(* CODESYS project IoDrvTemplate.library
   Version: 3.5.7.0
   Author: 3S - Smart Software Solutions GmbH
   Description: Template for an IO-driver written in IEC:
      Examples:
      - Bitfield
      - I/O Channels
      - Parameters
      - Diagnostic message and Acknowledge
      - Background diagnosis
      - CAA Device Diagnosis (incl. Reconfigure)
   Title: IoDrvTemplate
   DocFormat: reStructuredText
   DefaultNamespace: TPL
   LanguageModelAttribute: qualified-access-only
   Company: MyCompany
   Placeholder: IoDrvTemplate

Project tree, tasks and I/O mapping:
  libraries: SysMem, * (System); SysCpuHandling, * (System); IoDrvBase, * (System); IoStandard, * (System); IoDriver Parameter Interfaces, * (System); Base Interfaces, * (System); IoDriver Interfaces, * (System); CmpErrors2 Interfaces, * (System); SysTypes2 Interfaces, * (System); CAA Device Diagnosis, 3.5.8.0 (CAA Technical Workgroup); CAA Types Extern, * (CAA Technical Workgroup); CmpAsyncMgr, * (System)
  function block IoDrvTemplate [ST]: IoDrvWriteParameter, IoDrvReadParameter, IoDrvReadInputs, IoDrvIdentify, IoDrvUpdateConfiguration, IoDrvWatchdogTrigger, IoDrvScanModules, IoDrvUpdateMapping, IoDrvWriteOutputs, IoDrvStartBusCycle, IoDrvGetModuleDiagnosis, QueryInterface, FB_Reinit, Initialize, FB_Exit, FB_Init, IoDrvGetConnector, Cleanup, FreeScanData
  function block IoDrvTemplateDiag [ST]: ChildNodeCount, Connector, Enable, FirstChildNode, Index, IsRootNode, NextSiblingNode, ParentNode, SiblingNodeCount, GetChild, Initialize_Diag, GetSpecificDeviceState, SetCommunicationState, GetDeviceInfo, GetDeviceErrorAsync, GetSpecificDeviceErrorAsync, GetDeviceDiagnosisInfo, GetDeviceState, CheckCurrentSupportedCommunicationState, CheckSupportedCommunicationState, GetLogger, GetBusScanAsync, GetQoS, GetBusErrorAsync, GetBusDiagnosisInfo, GetBusState, GetBusInfo, GetSpecificBusState, ReconfigureActive, SiblingIRP, ReconfigureAsync, RegisterIRPChild
  Functions/
    function IsConnectorEnabled [ST]
  global variables GVL
*)

// GVL
VAR_GLOBAL
	g_stComponentName : STRING := 'IoDrvTemplate';
END_VAR

// IoDrvTemplate
{attribute 'no_assign'}
{attribute 'conditionalshow_all_locals' := 'IoDrvDebug'}
FUNCTION_BLOCK IoDrvTemplate EXTENDS IoDrvBase IMPLEMENTS ICmpIoDrvParameter
VAR_INPUT
END_VAR
VAR_OUTPUT
END_VAR
VAR CONSTANT
	CLASSID_CCmpIoDrvTemplate : DWORD := 16#0000FF02;
	IOSize : DWORD := 5;
END_VAR
VAR
	_byInputs : ARRAY [0..IOSize-1] OF BYTE;
	_byOutputs : ARRAY [0..IOSize-1] OF BYTE;
	_IIoDrv : ICmpIoDrv;
	_IIoDrvParameter : ICmpIoDrvParameter;
	_xBackGroundDiagStarted : BOOL;
	_bDeactivated : BOOL;
	
	//Variables for scan
	_iScannedSlaves : INT;
	_pScanList : POINTER TO IoStandard.IoConfigConnector;
END_VAR

{attribute 'conditionalshow' := 'IoDrvDebug'}
METHOD IoDrvWriteParameter : UDINT
VAR_INPUT
	pConnector : POINTER TO IoConfigConnector;
	pParameter : POINTER TO IoConfigParameter;
	pData : POINTER TO BYTE;
	dwBitSize : DWORD;
	dwBitOffset : DWORD;
END_VAR
VAR
	pParam : POINTER TO IoConfigParameter;
	pstDiagString : POINTER TO STRING;
	pValue : POINTER TO BYTE;
END_VAR
IF pConnector = 0 OR pParameter = 0 OR pData = 0 THEN
	IoDrvWriteParameter := Errors.ERR_PARAMETER;
	RETURN;	
END_IF

//If IoDrvWriteParameter returns a value unequal ERR_OK, write parameter will be handled by the IO-manager!
//Note: Code must be only implemented here if there are special things to do.

IoDrvWriteParameter := Errors.ERR_OK;

CASE pParameter^.dwParameterId OF
	393221: //simulate diag
		IF pData^ <> 0 THEN
			(*
				Example for extended Diagnostic:
				- here a string value is written to parameter of channeltype "diag": when "CF_CONNECTOR_DIAGNOSTIC_AVAILABLE" is set in the connector, the diagnostic message is read with ReadParameter.
			*)
			pParam := IoMgrConfigGetParameter(pConnector, 4711);
			IF pParam <> 0 THEN
				pstDiagString := IoMgrConfigGetParameterValuePointer(pParam, 0);
				IF pstDiagString <> 0 THEN
					pstDiagString^ := 'Error pending';
				END_IF
			END_IF
			
			(*
				set diagnostic available flag to trigger reading of diagnosis parameter
			*) 
			IoMgrConfigSetDiagnosis(pConnector, Connectorflags.CF_CONNECTOR_DIAGNOSTIC_AVAILABLE);
		END_IF
		RETURN;
	393222, 393223:
		//here you can add some special code for the three parameters
		pValue := pParameter^.dwValue;
		SysMemCpy((pValue + dwBitOffset/8), pData, MIN(DWORD_TO_BYTE(dwBitSize/8), UINT_TO_BYTE(pParameter^.wLen / 8)));			
		RETURN;
	4712: 
		(*
				Example for extended Diagnostic Acknowledge:
				- Parameter needs channel type "diagack": when user presses ACKNOWLEDGE WriteParameter is called
				- here only the flag is reset, so the diag message is not shown in the Editor any more  
		*)
		IoMgrConfigResetDiagnosis(pConnector, Connectorflags.CF_CONNECTOR_DIAGNOSTIC_AVAILABLE);
		RETURN;
	ELSE
		pValue := pParameter^.dwValue; 
		SysMemCpy(pDest := pValue + dwBitOffset/8, pSrc := pData, pParameter^.wLen / 8);
END_CASE

IoDrvWriteParameter := Errors.ERR_FAILED;
END_METHOD

{attribute 'conditionalshow' := 'IoDrvDebug'}
METHOD IoDrvReadParameter : UDINT
VAR_INPUT
	pConnector : POINTER TO IoConfigConnector;
	pParameter : POINTER TO IoConfigParameter;
	pData : POINTER TO BYTE;
	dwBitSize : DWORD;
	dwBitOffset : DWORD;
END_VAR
VAR
	pValue : POINTER TO BYTE;
END_VAR
IF 	pConnector = 0 OR pParameter = 0 OR pData = 0 THEN
	IoDrvReadParameter := Errors.ERR_PARAMETER;
	RETURN;	
END_IF

IoDrvReadParameter := Errors.ERR_OK;

pValue := pParameter^.dwValue;
IF pValue <> 0 THEN
	CASE pParameter^.dwParameterId OF
		4711: 
			(*
				Example for extended Diagnostic:
				- Parameter needs channel type "diag": as long as connectorflag "CF_CONNECTOR_DIAGNOSTIC_AVAILABLE" is set, the IoDrvReadParameter will be called with the Parameter of channeltype "diag"
				- One may return a string that is shown in "status" editor in CODESYS			
			*)

			IF pParameter^.wLen >= (dwBitOffset + dwBitSize) THEN	 
				SysMemCpy(pData, (pValue + dwBitOffset/8), MIN(DWORD_TO_BYTE(dwBitSize/8), UINT_TO_BYTE(pParameter^.wLen / 8)));		
				RETURN;
			END_IF
		ELSE
			// handle other parameters here: be aware of length of destination buffer
			SysMemCpy(pData, pValue + dwBitOffset/8, MIN(DWORD_TO_BYTE(dwBitSize/8), UINT_TO_BYTE(pParameter^.wLen / 8)));
			RETURN;
	END_CASE
END_IF
// All standard parameters of our device are handled by the IO-manager!
IoDrvReadParameter := Errors.ERR_FAILED;
END_METHOD

{attribute 'conditionalshow' := 'IoDrvDebug'}
METHOD IoDrvReadInputs : UDINT
VAR_INPUT
	pConnectorMapList : POINTER TO IoConfigConnectorMap;
	nCount : DINT;
END_VAR
VAR
	i,j : DINT;
	wSize : WORD;
	pConnectorMap : POINTER TO IoStandard.IoConfigConnectorMap;
	pChannelMap : POINTER TO IoStandard.IoConfigChannelMap;
	pbyIecAddress : POINTER TO BYTE;
	bySrcValue : BYTE;
	bySrcMask : BYTE;
	wSrcIndex : WORD;	
	wDestIndex : WORD;	
END_VAR
IoDrvReadInputs_Count := IoDrvReadInputs_Count + 1;

IF _bDeactivated THEN
	RETURN;
END_IF

IF pConnectorMapList = 0 OR nCount = 0 THEN
	IoDrvReadInputs := Errors.ERR_PARAMETER;
	RETURN;
END_IF

FOR i:=0 TO nCount - 1 DO
	pConnectorMap := ADR(pConnectorMapList[i]);
	
	FOR j:= 0 TO UDINT_TO_UINT(pConnectorMap^.dwNumOfChannels) - 1 DO
		pChannelMap := ADR(pConnectorMap^.pChannelMapList[j]);
		
		// input medium byteorder: Little Endian:		
		IoMgrCopyInputLE(pChannelMap, pChannelMap^.pParameter^.dwDriverSpecific);
		
		// input medium byteorder: Big Endian:		
		//IoMgrCopyInputBE(ADR(pChannelMap, pChannelMap^.pParameter^.dwDriverSpecific);
	END_FOR
END_FOR

IoDrvReadInputs := Errors.ERR_OK;
END_METHOD

{attribute 'conditionalshow' := 'IoDrvDebug'}
METHOD IoDrvIdentify : UDINT
VAR_INPUT
	pConnector : POINTER TO IoConfigConnector;	
END_VAR
VAR
END_VAR
IoDrvIdentify_Count := IoDrvIdentify_Count + 1;
IoDrvIdentify := Errors.ERR_NOTIMPLEMENTED;
END_METHOD

{attribute 'conditionalshow' := 'IoDrvDebug'}
METHOD IoDrvUpdateConfiguration : UDINT
VAR_INPUT
	pConnectorList : POINTER TO IoConfigConnector;
	nCount : DINT;
END_VAR
VAR
	pParameter : POINTER TO IoConfigParameter;	
	pChild : POINTER TO IoConfigConnector;	
	pstConnectorVendorName : POINTER TO STRING;
	pstConnectorDeviceName : POINTER TO STRING;
	dwTest : DWORD;
	Result : RTS_IEC_RESULT;
END_VAR
IoDrvUpdateConfiguration_Count := IoDrvUpdateConfiguration_Count + 1;
IoDrvUpdateConfiguration := Errors.ERR_OK;

IF pConnectorList = 0 THEN
	// Reset application
	m_pConnector^.hIoDrv := 0; // no callbacks from runtime!
	m_pConnector^.pFather^.hIoDrv := 0;
	Cleanup();
	RETURN;
END_IF

m_pConnector := IoMgrConfigGetConnector(pConnectorList, ADR(nCount), m_wModuleType, m_dwInstance);

IF m_pConnector = 0 THEN
	IoDrvUpdateConfiguration := ERRORS.ERR_PARAMETER;
	RETURN;
END_IF

//check if device is enabled in the device tree
_bDeactivated := NOT IsConnectorEnabled(m_pConnector);

IF m_pConnector^.hIoDrv = 0 THEN
	//always needed for reconfigure!
	m_pConnector^.hIoDrv := m_hInterface;
	m_pConnector^.pFather^.hIoDrv := m_hInterface;
END_IF

IF _bDeactivated THEN
	IoDrvUpdateConfiguration := CmpErrors.Errors.ERR_OK;
	RETURN;
END_IF

IF m_pConnector^.hIoDrv = m_hInterface THEN
	{IF defined (pou:IoMgrConfigSetDiagnosis)}
	IoMgrConfigSetDiagnosis(m_pConnector,
							ConnectorFlags.CF_DRIVER_AVAILABLE OR
							ConnectorFlags.CF_CONNECTOR_FOUND OR
							ConnectorFlags.CF_CONNECTOR_CONFIGURED OR
							ConnectorFlags.CF_CONNECTOR_ACTIVE);
	{END_IF}
	
	{IF defined (pou:IoMgrConfigSetDiagnosis)}
	IoMgrConfigSetDiagnosis(m_pConnector^.pFather,
							ConnectorFlags.CF_DRIVER_AVAILABLE OR
							ConnectorFlags.CF_CONNECTOR_FOUND OR
							ConnectorFlags.CF_CONNECTOR_CONFIGURED OR
							ConnectorFlags.CF_CONNECTOR_ACTIVE);
	{END_IF}

	{IF defined (pou:IoMgrSetDriverProperties)}			
		IoMgrSetDriverProperties(m_hInterface, DRVPROP_CONSISTENCY OR DRVPROP_BACKGROUND_GETDIAG);
		//Note: background diagnosis property flag is optional (supported with 3.5.1.0 runtime)
	{END_IF}										

	//Read some parameters
	pParameter := IoMgrConfigGetParameter(m_pConnector, 393218);
	IF pParameter <> 0 THEN
		pstConnectorVendorName := IoMgrConfigGetParameterValuePointer(pParameter, ADR(Result));
	END_IF
	pParameter := IoMgrConfigGetParameter(m_pConnector, 393219);
	IF pParameter <> 0 THEN
		pstConnectorDeviceName := IoMgrConfigGetParameterValuePointer(pParameter, ADR(Result));
	END_IF
	pParameter := IoMgrConfigGetParameter(m_pConnector, 393220);	(* test parameter *)
	IF (pParameter <> 0) THEN
		dwTest := IoMgrConfigGetParameterValueDword(pParameter, ADR(Result));	(* Test parameter value *)			
	END_IF
	
	//Setup I/O area
	pParameter := IoMgrConfigGetParameter(m_pConnector, 1000);		(* inputs *)
	IF (pParameter <> 0) THEN
		pParameter^.dwDriverSpecific := ADR(_byInputs[0]);					(* Device offset 0 *)
	END_IF
	pParameter := IoMgrConfigGetParameter(m_pConnector, 1001);		(* inputs *)
	IF (pParameter <> 0) THEN
		pParameter^.dwDriverSpecific := ADR(_byInputs[4]);					(* Device offset 0 *)
	END_IF
	pParameter := IoMgrConfigGetParameter(m_pConnector, 2000);		(* outputs *)
	IF (pParameter <> 0) THEN
		pParameter^.dwDriverSpecific := ADR(_byOutputs[0]);					(* Device offset 0 *)
	END_IF
	pParameter := IoMgrConfigGetParameter(m_pConnector, 2001);		(* outputs *)
	IF (pParameter <> 0) THEN
		pParameter^.dwDriverSpecific := ADR(_byOutputs[4]);					(* Device offset 0 *)
	END_IF
	
	//Go through all childs of the device
	pChild := IoMgrConfigGetFirstChild(m_pConnector, ADR(nCount), m_pConnector);
	WHILE (pChild <> 0) DO
		IF IsConnectorEnabled(pChild) THEN
			pChild^.hIoDrv := m_hInterface;	
			{IF defined (pou:IoMgrConfigSetDiagnosis)}
			IoMgrConfigSetDiagnosis(pChild,
									ConnectorFlags.CF_DRIVER_AVAILABLE OR
									ConnectorFlags.CF_CONNECTOR_FOUND OR
									ConnectorFlags.CF_CONNECTOR_CONFIGURED OR
									ConnectorFlags.CF_CONNECTOR_ACTIVE);
			{END_IF}
		END_IF
		pChild := IoMgrConfigGetNextChild(pChild, ADR(nCount), m_pConnector);
	END_WHILE
END_IF
END_METHOD

{attribute 'conditionalshow' := 'IoDrvDebug'}
METHOD IoDrvWatchdogTrigger : UDINT
VAR_INPUT
	pConnector : POINTER TO IoConfigConnector;	
END_VAR
VAR
END_VAR
IoDrvWatchdogTrigger_Count := IoDrvWatchdogTrigger_Count + 1;
IoDrvWatchdogTrigger := Errors.ERR_OK;
END_METHOD

{attribute 'conditionalshow' := 'IoDrvDebug'}
METHOD IoDrvScanModules : UDINT
VAR_INPUT
	pConnector : POINTER TO IoConfigConnector;
	ppConnectorList : POINTER TO POINTER TO IoConfigConnector;
	pnCount : POINTER TO DINT;	
END_VAR
VAR
	pCurConnector : POINTER TO IoConfigConnector;
	pParameter: POINTER TO IoConfigParameter;
	pString : POINTER TO STRING;
	i : INT;
	j : INT;
END_VAR
IoDrvScanModules_Count := IoDrvScanModules_Count + 1;

IF pConnector = 0 OR ppConnectorList = 0 OR pnCount = 0 THEN
	IoDrvScanModules := Errors.ERR_PARAMETER;
	RETURN;
END_IF

FreeScanData();

pnCount^ := 0;
ppConnectorList^ := 0;

(*
	TODO: implement specific bus scan!
	Note: IoDrvScanModules is called in communication task. If this method takes too long (> 20s) a communication timeout may happen.
	In this cases you can do a segmented scan by setting IoStandard.ConnectorOptions.CO_SCAN_PENDING_SUPPORTED.
	If IoDrvScanModules returns ERR_PENDING method is called again. The results of all calls are combined by the GUI.
*)

(*The following code just generates some example data. The real scan algorithm has to set the values regarding to the scan result. *)
_iScannedSlaves := 2; //we return 2 slaves

IF _iScannedSlaves > 0 THEN
	//Allocate memory for the connector list
	ppConnectorList^ := SysMemAllocData(g_stComponentName, INT_TO_DWORD(_iScannedSlaves * SIZEOF(IoStandard.IoConfigConnector)), 0);
	IF ppConnectorList = 0 THEN
		IoDrvScanModules := Errors.ERR_FAILED;
		_iScannedSlaves := 0;
		RETURN;
	END_IF
	SysMem.SysMemSet(ppConnectorList^, 0, INT_TO_DWORD(_iScannedSlaves * SIZEOF(IoStandard.IoConfigConnector)));
END_IF

pCurConnector := ppConnectorList^;
FOR i := 0 TO _iScannedSlaves - 1 DO
	pCurConnector^.dwNumOfParameters := 4; //we return the 4 mandatory parameters
	//Alocate memory for the parameter list of the current connector
	pCurConnector^.pParameterList := SysMemAllocData(g_stComponentName, pCurConnector^.dwNumOfParameters * SIZEOF(IoStandard.IoConfigParameter), 0);
	SysMem.SysMemSet(pCurConnector^.pParameterList, 0, pCurConnector^.dwNumOfParameters * SIZEOF(IoStandard.IoConfigParameter));
	
    pParameter := pCurConnector^.pParameterList;
	
	//Set parameter: Vendor code
	pParameter^.dwParameterId := 1;
	pParameter^.dwValue := 1; //Vendor Code
	pParameter^.wLen := 32;
	pParameter^.wType := INT_TO_WORD(TypeClass.TYPE_DWORD); //16#4
	pParameter^.dwFlags := IoStandard.PVF_READ OR IoStandard.PVF_WRITE OR IoStandard.PVF_VALUE; //16#34
	
	pParameter := pParameter + SIZEOF(IoStandard.IoConfigParameter);
	
	//Set parameter: Product code
	pParameter^.dwParameterId := 2;
	pParameter^.dwValue := 2; //Product Code
	pParameter^.wLen := 32;
	pParameter^.wType := INT_TO_WORD(TypeClass.TYPE_DWORD); //16#4
	pParameter^.dwFlags := IoStandard.PVF_READ OR IoStandard.PVF_WRITE OR IoStandard.PVF_VALUE; //16#34
	
	pParameter := pParameter + SIZEOF(IoStandard.IoConfigParameter);
	
	//Set parameter: Revision Number
	pParameter^.dwParameterId := 3;
	pParameter^.dwValue := 10; //Revision Number
	pParameter^.wLen := 32;
	pParameter^.wType := INT_TO_WORD(TypeClass.TYPE_DWORD); //16#4
	pParameter^.dwFlags := IoStandard.PVF_READ OR IoStandard.PVF_WRITE OR IoStandard.PVF_VALUE; //16#34
	
	pParameter := pParameter + SIZEOF(IoStandard.IoConfigParameter);
	
	//Set parameter: Device Identification
	pParameter^.dwParameterId := 4;
	pParameter^.dwValue := SysMemAllocData(g_stComponentName, SIZEOF(STRING), 0);
	pString := pParameter^.dwValue;
	pString^ := '1_2_10'; // Device Identification
	pParameter^.wLen := SIZEOF(STRING);
	pParameter^.wType := INT_TO_WORD(TypeClass.TYPE_STRING); //16#10
	pParameter^.dwFlags := IoStandard.PVF_READ OR IoStandard.PVF_WRITE OR IoStandard.PVF_POINTER; //16#32
		
	pCurConnector^.hIoDrv := THIS;
	pCurConnector^.pFather := pConnector;
	pCurConnector^.wType := ConnectorTypes.CT_CAN_SLAVE; //we return a CANopen Slave connector
	
	pCurConnector := pCurConnector + SIZEOF(IoStandard.IoConfigConnector);
END_FOR

pnCount^ := _iScannedSlaves; //Set number of scanned devices
IoDrvScanModules := CmpErrors.Errors.ERR_OK;
END_METHOD

{attribute 'conditionalshow' := 'IoDrvDebug'}
METHOD IoDrvUpdateMapping : UDINT
VAR_INPUT
	pTaskMapList : POINTER TO IoConfigTaskMap;
	nCount : DINT;	
END_VAR
VAR
END_VAR
IoDrvUpdateMapping_Count := IoDrvUpdateMapping_Count + 1;

IF (pTaskMapList = 0) THEN
	IoDrvUpdateMapping := Errors.ERR_PARAMETER;
	RETURN;
END_IF

IoDrvUpdateMapping := Errors.ERR_OK;
END_METHOD

{attribute 'conditionalshow' := 'IoDrvDebug'}
METHOD IoDrvWriteOutputs : UDINT
VAR_INPUT
	pConnectorMapList : POINTER TO IoConfigConnectorMap;
	nCount : DINT;
END_VAR
VAR
	i,j : DINT;
	wSize : WORD;
	pConnectorMap : POINTER TO IoStandard.IoConfigConnectorMap;
	pChannelMap : POINTER TO IoStandard.IoConfigChannelMap;
	pbyIecAddress : POINTER TO BYTE;
	bySrcValue : BYTE;
	wSrcIndex : WORD;	
	bySrcMask : BYTE;
	wDestIndex : WORD;	
END_VAR
IoDrvWriteOutputs_Count := IoDrvWriteOutputs_Count + 1;

IF _bDeactivated THEN
	RETURN;
END_IF

IF pConnectorMapList = 0 OR nCount = 0 THEN
	IoDrvWriteOutputs := Errors.ERR_PARAMETER;
	RETURN;
END_IF

FOR i:=0 TO nCount - 1 DO
	pConnectorMap := ADR(pConnectorMapList[i]);
	
	FOR j:= 0 TO UDINT_TO_UINT(pConnectorMap^.dwNumOfChannels) - 1 DO
		pChannelMap := ADR(pConnectorMap^.pChannelMapList[j]);
		
		// output medium byteorder: Little Endian:		
		IoMgrCopyOutputLE(pChannelMap, pChannelMap^.pParameter^.dwDriverSpecific);
		
		// output medium byteorder: Big Endian:		
		//IoMgrCopyOutputBE(pChannelMap, pChannelMap^.pParameter^.dwDriverSpecific);
	END_FOR
END_FOR

IoDrvWriteOutputs := Errors.ERR_OK;
END_METHOD

{attribute 'conditionalshow' := 'IoDrvDebug'}
METHOD IoDrvStartBusCycle : UDINT
VAR_INPUT
	pConnector : POINTER TO IoConfigConnector;
END_VAR
VAR
END_VAR
IoDrvStartBusCycle_Count := IoDrvStartBusCycle_Count + 1;

IF _bDeactivated OR_ELSE pConnector <> m_pConnector THEN
	RETURN;
END_IF

//if background diagnosis is not active call IoDrvGetModuleDiagnosis; normally it will be called by the runtime if DRVPROP_BACKGROUND_GETDIAG is set
IF NOT _xBackGroundDiagStarted THEN
	IoDrvGetModuleDiagnosis(m_pConnector); //DRVPROP_BACKGROUND_GETDIAG not set or runtime version < V3.5.1.0
END_IF

//optional: call IoDrvWatchdogTrigger or set driver property DRVPROP_WATCHDOG in UpdateConfiguration
IoDrvWatchdogTrigger(pConnector);

//simulate input data (only for test)
MemCpy(ADR(_byInputs), ADR(_byOutputs), IOSize);

IoDrvStartBusCycle := Errors.ERR_OK;
END_METHOD

METHOD IoDrvGetModuleDiagnosis : UDINT
VAR_INPUT
	pConnector : POINTER TO IoConfigConnector;
END_VAR
VAR
END_VAR
IF pConnector = 0 THEN
	//we are called from the background task
	_xBackGroundDiagStarted := TRUE;
END_IF

//Todo: update connectorflags if something changed

IoDrvGetModuleDiagnosis_Count := IoDrvGetModuleDiagnosis_Count + 1;
IoDrvGetModuleDiagnosis := Errors.ERR_NOTIMPLEMENTED;
END_METHOD

{attribute 'conditionalshow' := 'IoDrvDebug'}
METHOD QueryInterface : POINTER TO POINTER TO BYTE
VAR_INPUT
	iid : DWORD; (* InterfaceID *)
	pResult : POINTER TO UDINT;	
END_VAR
VAR
END_VAR
QueryInterface_Count := QueryInterface_Count + 1;
IF iid = ITFID_ICmpIoDrv THEN
	QueryInterface := ADR(_IIoDrv);
	AddRef();
	IF (pResult <> 0) THEN
		pResult^ := Errors.ERR_OK;
	END_IF
	RETURN;	
ELSIF iid = ITFID_ICmpIoDrvParameter THEN
	QueryInterface := ADR(_IIoDrvParameter);
	AddRef();
	IF (pResult <> 0) THEN
		pResult^ := Errors.ERR_OK;
	END_IF	
	RETURN;	
ELSE
	QueryInterface := SUPER^.QueryInterface(iid, pResult);
END_IF
END_METHOD

{attribute 'conditionalshow' := 'IoDrvDebug'}
METHOD FB_Reinit : BOOL
VAR_INPUT
END_VAR
VAR
END_VAR
FB_Reinit_Count := FB_Reinit_Count + 1;
FB_Reinit := TRUE;
END_METHOD

{attribute 'conditionalshow' := 'IoDrvDebug'}
METHOD Initialize : UDINT
VAR_INPUT
	wModuleType : UINT;
	dwInstance : UDINT;
	pConnector : POINTER TO IoConfigConnector; 
END_VAR
VAR
END_VAR
Initialize_Count := Initialize_Count + 1;

m_wModuleType := wModuleType;
m_dwInstance := dwInstance;
m_Info.wModuleType := wModuleType;

Initialize := Errors.ERR_OK;
END_METHOD

{attribute 'conditionalshow' := 'IoDrvDebug'}
METHOD FB_Exit : BOOL
VAR_INPUT
	bInCopyCode: BOOL;	
END_VAR
VAR
END_VAR
FB_Exit_Count := FB_Exit_Count + 1;
FB_Exit := TRUE;
END_METHOD

{attribute 'conditionalshow' := 'IoDrvDebug'}
METHOD FB_Init : BOOL
VAR_INPUT
	bInitRetains: BOOL;
	bInCopyCode: BOOL;
END_VAR
VAR
	Result : UDINT;
END_VAR
FB_Init_Count := FB_Init_Count + 1;

m_Info.szDriverName := 'IoDrvTemplateIEC';
m_Info.szVendorName := 'MyCompany';
m_Info.szDeviceName := 'MyCard';
m_Info.wModuleType := 40100;

_IIoDrv := THIS^;
_IIoDrvParameter := THIS^;

m_IBaseItf := THIS^;
m_hInterface := IoMgrRegisterInstance2(CLASSID_CCmpIoDrvTemplate, m_IBaseItf, ADR(Result));
FB_Init := TRUE;
END_METHOD

{attribute 'conditionalshow' := 'IoDrvDebug'}
METHOD IoDrvGetConnector : POINTER TO IoConfigConnector
VAR_INPUT
	pResult : POINTER TO RTS_IEC_RESULT;
END_VAR
VAR
END_VAR
IF m_pConnector = 0 THEN
	IF pResult <> 0 THEN
		pResult^ := Errors.ERR_FAILED;
	END_IF
	IoDrvGetConnector := 0;	
	RETURN;
END_IF
IF pResult <> 0 THEN
	pResult^ := Errors.ERR_OK;
END_IF
IoDrvGetConnector := m_pConnector;
END_METHOD

{attribute 'conditionalshow' := 'IoDrvDebug'}
METHOD Cleanup
VAR_INPUT
END_VAR
VAR

END_VAR
FreeScanData();
END_METHOD

{attribute 'conditionalshow' := 'IoDrvDebug'}
METHOD FreeScanData
VAR_INPUT
END_VAR
VAR
	pCurConnector : POINTER TO IoConfigConnector;
	pParameter : POINTER TO IoConfigParameter;	
	i : INT;
	j : INT;
END_VAR
//Free device scan data
IF _iScannedSlaves > 0 AND _pScanList <> 0 THEN
	pCurConnector := _pScanList;
	FOR i := 0 TO _iScannedSlaves - 1 DO
		pParameter := pCurConnector^.pParameterList;
		IF pParameter <> 0 THEN
			FOR j := 0 TO DWORD_TO_INT(pCurConnector^.dwNumOfParameters) - 1 DO
				IF (pParameter^.dwFlags AND IoStandard.ParameterValueFlags.PVF_POINTER) = IoStandard.ParameterValueFlags.PVF_POINTER THEN
					// dwValue is pointer
					IF pParameter^.dwValue <> 0 THEN
						SysMemFreeData(g_stComponentName, pParameter^.dwValue);
					END_IF
				END_IF
				pParameter := pParameter + SIZEOF(IoConfigParameter);	
			END_FOR
			SysMemFreeData(g_stComponentName, pCurConnector^.pParameterList);
		END_IF
		pCurConnector := pCurConnector + SIZEOF(IoStandard.IoConfigConnector);
	END_FOR
	SysMemFreeData(g_stComponentName, _pScanList);
	_pScanList := 0;
 	_iScannedSlaves := 0;
END_IF
END_METHOD

END_FUNCTION_BLOCK

// Functions/IsConnectorEnabled
{attribute 'conditionalshow' := '3SLib_Developer'}
FUNCTION IsConnectorEnabled : BOOL
VAR_INPUT
	pConnector : POINTER TO IoStandard.IoConfigConnector;
END_VAR
VAR
END_VAR

{IF defined (variable:CF_DEVICE_ENABLED) AND defined (variable:CF_DIAG_PROVIDER)}
	IF (pConnector^.dwFlags AND IoStandard.ConnectorFlags.CF_DIAG_PROVIDER) <> 0 THEN
		IsConnectorEnabled := (pConnector^.dwFlags AND IoStandard.ConnectorFlags.CF_DEVICE_ENABLED) <> 0;
	ELSE
		IsConnectorEnabled := (pConnector^.dwFlags AND ConnectorFlags.CF_ENABLE) <> 0;
	END_IF
{ELSE}
	IsConnectorEnabled := (pConnector^.dwFlags AND ConnectorFlags.CF_ENABLE) <> 0;
{END_IF}

END_FUNCTION

// IoDrvTemplateDiag
//This function block implements the diagnosis code for CAA Device Diagnosis.
{attribute 'no_assign'}
{attribute 'conditionalshow_all_locals' := 'IoDrvDebug'}
FUNCTION_BLOCK IoDrvTemplateDiag EXTENDS IoDrvTemplate IMPLEMENTS DED.IDevice2, DED.IBus, DED.IStack, DED.IReconfigureProvider
VAR_INPUT
END_VAR
VAR_OUTPUT
END_VAR
VAR
	_diag : DED.CAADiagnosisBase;
	_tree : DED.CAADiagTreeBase;
	_reconfig : DED.CAAReconfigureBase; //optional
END_VAR

(*Returns the number of childs below the current node*)
PROPERTY ChildNodeCount : CAA.COUNT
GET
ChildNodeCount := _tree.ChildNodeCount;
END_GET
END_PROPERTY

PROPERTY Connector : POINTER TO IoStandard.IoConfigConnector
GET
Connector := _tree.Connector;
END_GET
END_PROPERTY

(*This property returns if the node is enabled in the device tree. The setter can be used to change the Enabled flag. If enabling/disabling is not supported on the node the flag’s value will not change.*)
PROPERTY Enable : BOOL
GET
Enable := _tree.Enable;
END_GET
SET
_tree.Enable := Enable;
END_SET
END_PROPERTY

(*Returns the first child node below the current one*)
PROPERTY FirstChildNode : DED.INode
GET
FirstChildNode := _tree.FirstChildNode;
END_GET
END_PROPERTY

PROPERTY Index : UDINT
GET
Index := _tree.Index;
END_GET
SET
_tree.Index := Index;
END_SET
END_PROPERTY

(* returns true, if the current node is the root (plc) node, otherwise false*)
PROPERTY IsRootNode : BOOL
GET
IsRootNode := _tree.IsRootNode;
END_GET
END_PROPERTY

(* returns the next sibling node at the same level
 used for step through all nodes*)
PROPERTY NextSiblingNode : DED.INode
GET
NextSiblingNode := _tree.NextSiblingNode;
END_GET
END_PROPERTY

(* Returns the parent node or zero if already the root node is reached*)
PROPERTY ParentNode : DED.INode
GET
ParentNode := _tree.ParentNode;
END_GET
END_PROPERTY

(* Returns the number of sibling (same level) nodes*)
PROPERTY SiblingNodeCount : CAA.COUNT
GET
SiblingNodeCount := _tree.SiblingNodeCount;
END_GET
END_PROPERTY

{attribute 'hide'}
METHOD GetChild : DED.INode
VAR_INPUT
	udiIndex	: UDINT;
END_VAR
GetChild:= _tree.GetChild(udiIndex);
END_METHOD

{attribute 'hide'}
METHOD Initialize_Diag : UDINT
VAR_INPUT
	pConnector	: POINTER TO IoStandard.IoConfigConnector;
	nConnectorCount	: DINT;
	parent	: POINTER TO DED.INode;
	children	: POINTER TO DED.INode;
	udiChildCount	: UDINT;
END_VAR
//general initialization code: do not remove!
_tree.Initialize_Diag(pConnector, nConnectorCount, parent, children, udiChildCount);
_diag.Initialize_Diag(pConnector, nConnectorCount);

//if IReconfigureProvider is implemented
_reconfig.Initialize_Diag(THIS^);
END_METHOD

{attribute '''NORMAL__COMMENT' := 'Returns the fieldbus specific device state; interpretation is fieldbus dependent'}
(*Returns the fieldbus specific device state; interpretation is fieldbus dependent*)
METHOD GetSpecificDeviceState : DED.ERROR (* eError *)
VAR_INPUT
	(*Pointer to memory*)
	pData	: CAA.PVOID;
	(*Size of memory in bytes where pData is pointing to*)
	szSize	: CAA.SIZE;
END_VAR
VAR_OUTPUT
	(*Number of Bytes written to pData*)
	szCount	: CAA.SIZE;
END_VAR
GetSpecificDeviceState := DED.ERROR.NOT_SUPPORTED;
END_METHOD

(*Starts, stops or resets a device*)
METHOD SetCommunicationState : DED.ERROR (* eError *)
VAR_INPUT
	eRequestedState	: DED.DEVICE_TRANSITION_STATE;
END_VAR
IF CheckCurrentSupportedCommunicationState(eRequestedState) THEN
	CASE eRequestedState OF
		DED.DEVICE_TRANSITION_STATE.RESET:
			//TODO: Send a reset command to the device.
		DED.DEVICE_TRANSITION_STATE.START:
			//TODO: Send a start command to the device.
		DED.DEVICE_TRANSITION_STATE.STOP:
			//TODO: Send a stop command to the device.
	END_CASE
ELSE
	SetCommunicationState := DED.ERROR.OPERATION_INVALID;
END_IF
END_METHOD

(*Returns the device information of the current node*)
METHOD GetDeviceInfo : DED.ERROR (*eError*)
VAR_IN_OUT
	(*Device information struct*)
	deiInfo	: DED.DEVICE_INFO;
END_VAR
//base implementation supports all 3S specific fieldbusses.
GetDeviceInfo := _diag.GetDeviceInfo(deiInfo);
END_METHOD

{attribute 'hide'}
(* Returns the device error of the current node; you can also use functionblock GetDeviceError.*)
METHOD GetDeviceErrorAsync : DED.PROC_STATE (* eState *)
VAR_INPUT
	(*eCommand*)
	eCmd	: DED.PROC_CMD;
END_VAR
VAR_IN_OUT
	(*error struct*)
	eriDeviceError	: DED.ERROR_INFO;
END_VAR
VAR_OUTPUT
	(*error code if method fails*)
	eError	: DED.ERROR;
END_VAR
//optional method; base implementation returns NOT_SUPPORTED
GetDeviceErrorAsync := _diag.GetErrorAsync(eCmd, eriDeviceError, eError => eError);
END_METHOD

{attribute 'hide'}
(*Returns the specific device error of the current node; interpretation is fieldbus-dependent; you can also use functionblock GetSpecificDeviceError*)
METHOD GetSpecificDeviceErrorAsync : DED.PROC_STATE (* eState *)
VAR_INPUT
	(*eCommand*)
	eCmd	: DED.PROC_CMD;
	(*Pointer to memory*)
	pData	: CAA.PVOID;
	(*Size of memory in bytes where pData is pointing to*)
	szSize	: CAA.SIZE;
END_VAR
VAR_OUTPUT
	(*Number of Bytes written to pData*)
	szCount	: CAA.SIZE;
	(*error code if method fails*)
	eError	: DED.ERROR;
END_VAR
//optional method; base implementation returns NOT_SUPPORTED
GetSpecificDeviceErrorAsync := _diag.GetSpecificDeviceErrorAsync(eCmd,pData, szSize, szCount=>szCount, eError => eError);
END_METHOD

{attribute '''NORMAL__COMMENT' := 'Returns a DiagnosisInfo if xDiagnosisInfoAvailable of GetDeviceState was true.'}
(*Returns a DiagnosisInfo if xDiagnosisInfoAvailable of GetDeviceState was true.*)
METHOD GetDeviceDiagnosisInfo : DED.ERROR (*eError*)
VAR_INPUT
	(*Pointer to memory*)
	pData	: CAA.PVOID;
	(*Size of memory in bytes where pData is pointing to*)
	szSize	: CAA.SIZE;
END_VAR
VAR_OUTPUT
	(*Number of Bytes written to pData*)
	szCount	: CAA.SIZE;
END_VAR
//This is an optional method. Return device specific diagnostic information
GetDeviceDiagnosisInfo := DED.ERROR.NOT_SUPPORTED;
END_METHOD

(*Returns the state of the device; if device state is ERROR further information can be read by GetDeviceError*)
METHOD GetDeviceState : DED.DEVICE_STATE (* eDeviceState *)
VAR_OUTPUT
	(*if true, diagnosis info can be read by calling GetDeviceDiagnosisInfo*)
	xDiagnosisInfoAvailable	: BOOL;
	eError	: DED.ERROR;
END_VAR
//base implementation reads connector flags and delivers the right state
GetDeviceState := _diag.GetState(xDiagnosisInfoAvailable => xDiagnosisInfoAvailable, eError => eError);

//Sometimes you want to overload the connector flags state. Then use additionaly the following code.
IF GetDeviceState <> DED.DEVICE_STATE.DISABLED THEN
	IF GetBusState() = DED.BUS_STATE.ERROR THEN
		GetDeviceState := DED.DEVICE_STATE.ERROR;
	ELSE
		//TODO: return specific state
	END_IF
END_IF
END_METHOD

(* Returns true if the driver in the current state supports the requested communications state
 The method CheckSupportedCommunicationState is used to check for the general availability of communications states
 Therefore the result of CheckCurrentSupportedCommunicationState and CheckSupportedCommunicationState could differ if the driver is for example in the startup procedure and
 not supporting currently some communication states.*)
METHOD CheckCurrentSupportedCommunicationState : BOOL (* True, if state is supported*)
VAR_INPUT
	(* The communication state to check *)
	eRequestedState	: DED.DEVICE_TRANSITION_STATE;
END_VAR
CheckCurrentSupportedCommunicationState := (GetDeviceState() <> DED.DEVICE_STATE.DISABLED) AND CheckSupportedCommunicationState(eRequestedState);
END_METHOD

(* The implementation of this method returns true if the driver supports the requested communications state
 The application could query a driver to check if it is supporting specific communications states generally.
 The method CheckCurrentSupportedCommunicationState is used to check for the current state.
 Therefore the result of CheckCurrentSupportedCommunicationState and CheckSupportedCommunicationState could differ if the driver is for example in the startup procedure and
 not supporting currently some communication states.*)
METHOD CheckSupportedCommunicationState : BOOL (* True, if state is supported*)
VAR_INPUT
	(* The communication state to check *)
	eRequestedState	: DED.DEVICE_TRANSITION_STATE;
END_VAR
CASE eRequestedState OF
	DED.DEVICE_TRANSITION_STATE.RESET, DED.DEVICE_TRANSITION_STATE.START, DED.DEVICE_TRANSITION_STATE.STOP:
		CheckSupportedCommunicationState := TRUE;
END_CASE
END_METHOD

METHOD GetLogger : DED.ILogger
VAR_OUTPUT
	eError	: DED.ERROR;
END_VAR
eError := DED.ERROR.NOT_SUPPORTED;
END_METHOD

{attribute '''NORMAL__COMMENT' := 'Returns the bus scan of the current node'}
(*Returns the bus scan of the current node*)
METHOD GetBusScanAsync : DED.PROC_STATE
VAR_INPUT
	(*eCommand*)
	eCmd	: DED.PROC_CMD;
END_VAR
VAR_OUTPUT
	(* First node of scanned device list*)
	itfFirstDevice	: DED.INode;
	eError	: DED.ERROR;
END_VAR
//optional method; base implementation returns NOT_SUPPORTED
GetBusScanAsync := _diag.GetBusScanAsync(eCmd);
END_METHOD

METHOD GetQoS : DED.ERROR
VAR_IN_OUT
	QualityInfo	: DED.QOS_INFO;
END_VAR
//TODO: Return quality of service informations e.g. busload, error counter,...
GetQoS := DED.ERROR.NOT_SUPPORTED;
END_METHOD

{attribute 'hide'}
(*Returns the bus error of the current node; you can also use functionblock GetBusError.*)
METHOD GetBusErrorAsync : DED.PROC_STATE (* eState *)
VAR_INPUT
	(*eCommand*)
	eCmd : DED.PROC_CMD;
END_VAR
VAR_IN_OUT
	(*error struct*)
	eriBusError	: DED.ERROR_INFO;
END_VAR
VAR_OUTPUT
	eError	: DED.ERROR;
END_VAR
//optional method; base implementation returns NOT_SUPPORTED
GetBusErrorAsync := _diag.GetErrorAsync(eCmd := eCmd, eriError := eriBusError, eError => eError);
END_METHOD

(*Returns a DiagnosisInfo if xDiagnosisInfoAvailable of GetBusState was true.*)
METHOD GetBusDiagnosisInfo : DED.ERROR (* eError *)
VAR_INPUT
	(*Pointer to memory*)
	pData	: CAA.PVOID;
	(*Size of memory in bytes where pData is pointing to*)
	szSize	: CAA.SIZE;
END_VAR
VAR_OUTPUT
	(*Number of Bytes written to pData*)
	szCount	: CAA.SIZE;
END_VAR
//This is an optional method. Return bus specific diagnostic information
GetBusDiagnosisInfo := DED.ERROR.NOT_SUPPORTED;
END_METHOD

(*Returns the bus state of the current node; if device state is ERROR further information can be read by GetBusError*)
METHOD GetBusState : DED.BUS_STATE (* eBusState *)
VAR_OUTPUT
	(*if true, diagnosis info can be read by calling GetBusDiagnosisInfo*)
	xDiagnosisInfoAvailable	: BOOL;
	eError	: DED.ERROR;
END_VAR
//base implementation reads connector flags and delivers the right state
GetBusState := _diag.GetBusState(xDiagnosisInfoAvailable => xDiagnosisInfoAvailable, eError => eError);

//Sometimes you want to overload the connector flags state. Then use additionaly the following code.
IF GetBusState <> DED.BUS_STATE.DISABLED THEN //if not disabled
	//TODO: return specific bus state 
END_IF
END_METHOD

(*Returns the bus information of the current node*)
METHOD GetBusInfo : DED.ERROR (*eError*)
VAR_IN_OUT
	(*Bus information struct*)
	buiInfo	: DED.BUS_INFO;
END_VAR
//base implementation supports all 3S specific fieldbusses.
GetBusInfo := _diag.GetBusInfo(buiInfo);
END_METHOD

(*Returns the fieldbus specific bus state; interpretation is fieldbus dependent*)
METHOD GetSpecificBusState : DED.ERROR (* eError *)
VAR_INPUT
	(*Pointer to memory*)
	pData	: CAA.PVOID;
	(*Size of memory in bytes where pData is pointing to*)
	szSize	: CAA.SIZE;
END_VAR
VAR_OUTPUT
	(*Number of Bytes written to pData*)
	szCount	: CAA.SIZE;
END_VAR
GetSpecificBusState := DED.ERROR.NOT_SUPPORTED;
END_METHOD

(* This property is TRUE if reconfiguration is currently active.*)
{attribute 'conditionalshow' := '3SLib_Developer'}
PROPERTY ReconfigureActive : BOOL
GET
ReconfigureActive := _reconfig.ReconfigureActive;
END_GET
END_PROPERTY

(* Gets and sets the next sibling IReconfigureProvider.*)
{attribute 'conditionalshow' := '3SLib_Developer'}
PROPERTY SiblingIRP : DED.IReconfigureProvider
GET
SiblingIRP := _reconfig.SiblingIRP;
END_GET
SET
_reconfig.SiblingIRP := SiblingIRP;
END_SET
END_PROPERTY

(* Reconfigure reads the configuration of the corresponding node and applies it.
 Afterwards it calls ReconfigureAsync for all child IReconfigureProvider.
 After Reconfiguring all changed configuration values (Enable flag, Parameter changes,...) take effect.
 If the node doesn't support reconfiguring, method returns ERROR and eError contains |ERROR.NOT_SUPPORTED|.*)
 {attribute 'conditionalshow' := '3SLib_Developer'}
METHOD ReconfigureAsync : DED.PROC_STATE
VAR_INPUT
	(*eCommand: EXECUTE to start operation.*)
	eCmd	: DED.PROC_CMD;
	(*Originator of reconfiguration. 0 or current node if this is the first reconfiguration call.*)
	itfSender	: DED.INode;
END_VAR
VAR_OUTPUT
	(*Error code*)
	eError	: DED.ERROR;
END_VAR
//This method is used by CAA Device Diagnosis Reconfigure function block.
//The following example uses the reconfigure base implementation for I/O drivers. First it calls _reconfig.ReconfigureIoDriverAsync which uses IoStandard.IoMgrReconfigure.
//IoMgrReconfigure triggers a complete asynchronous reinitialization of the corresponding I/O driver 
//(IoDrvUpdateConfiguration with 0, IoDrvUpdatConfiguration with connectorlist and IoDrvUpdateMapping).
//Afterwards _reconfig.ReconfigureChildrenAsync is called which does a reconfigure on all children implementing IReconfigurationProvider. 
//For this it's necessary that _reconfig.Initialize_Diag is called in INode.Initialize_Diag!
//
//Note: It's also possible to implement Reconfigure in a different way e.g. if a stack supports Reconfigure for single child devices.
//In this case functionblocks for child devices have to implement IReconfigureProvider as well.

ReconfigureAsync := _reconfig.ReconfigureAsync(eCmd, itfSender, eError => eError);

(* CODE SNIPPET for custom specific implementation
{IF defined (pou:IoMgrReconfigure) AND defined (variable:ASYNCSTATE_READY)}
	CASE eCmd OF
		DED.PROC_CMD.EXECUTE:
			IF _byReconfigureState = 0 THEN
				IF itfSender = 0 THEN //if itfSender is current node ==> we are the originator; if someone calls us with 0, we also assume we are the originator.
					itfSender := THIS^; 
				END_IF
				
				_reconfig.BeginReconfigure(itfSender); //begin reconfiguration: if this is the first reconfigure call ==> enable flags are updated
				
				_xReconfigureError := FALSE; //member variable for memorizing errors
				_byReconfigureState := 1;
			END_IF
			
			IF _byReconfigureState = 1 THEN
				//TODO: Execute specific code
				//e.g. eProcState := ReconfigureNodeAsync(itfSender)
				IF eProcState = DED.PROC_STATE.DONE OR eProcState = DED.PROC_STATE.ERROR THEN
					_xReconfigureError := _xReconfigureError OR (eProcState = DED.PROC_STATE.ERROR);
					_byReconfigureState := 2;
				END_IF
			END_IF
			
			IF _byReconfigureState = 2 THEN
				//delegate reconfigure to all children implementing IReconfigureProvider (children are registered in Initialize_Diag by base implementation)
				eProcState := ReconfigureChildrenAsync(eCmd, itfSender);
				IF eProcState = DED.PROC_STATE.DONE OR eProcState = DED.PROC_STATE.ERROR THEN
					_xReconfigureError := _xReconfigureError OR (eProcState = DED.PROC_STATE.ERROR);
					_byReconfigureState := 0;
				END_IF
			END_IF

			IF _byReconfigureState <> 0 THEN
				ReconfigureAsync := DED.PROC_STATE.BUSY;
			ELSE
				IF _xReconfigureError THEN
					ReconfigureAsync := DED.PROC_STATE.ERROR;
					eError := DED.ERROR.ERROR_IO;
				ELSE
					ReconfigureAsync := DED.PROC_STATE.DONE;
				END_IF
				
				_reconfig.EndReconfigure(itfSender); //end reconfiguration
			END_IF
		ELSE
			//unexpected eCmd
			eError := DED.ERROR.PARAM_INVALID;
			ReconfigureAsync := DED.PROC_STATE.ERROR;
END_CASE
{ELSE}
	//old IoStandard library ==> reconfigure not supported
	ReconfigureAsync := DED.PROC_STATE.ERROR;
	eError := DED.ERROR.NOT_SUPPORTED;
{END_IF}
*)
END_METHOD

(* This method is used by IReconfigureProvider children to register at their parent.*)
{attribute 'conditionalshow' := '3SLib_Developer'}
METHOD RegisterIRPChild : DED.ERROR
VAR_INPUT
	itfChild	: DED.IReconfigureProvider;
END_VAR
RegisterIRPChild := _reconfig.RegisterIRPChild(itfChild);
END_METHOD

END_FUNCTION_BLOCK
